(* PLC project Untitled1, Beckhoff Automation GmbH TwinCAT PLC Control 3.5.13.21 *)
(* stored: creationDateTime 2024-03-06T00:00:47.2111878, modificationDateTime 2024-03-06T00:00:47.2111878 *)

PROGRAM main_1
VAR
//Problem1: Start from input1, go clockwise(out1) reset from input 3. To have sufficient time to stop, the Reset button will remain 
//active for 3s from Tof_0. The condition to reset out1 is that out1 has to be active, and out2 has to deactivate. 
//The condition to active out1 is out2 has to deactivate, reset for out1 and out2 has to deactive. The same thing for out2 go for counterclockwise


//Problem2 :Start from input1, it will active Tof_2 for 5 seconds -> run out1 from RS_0 for 5 seconds. And out1 connect to ToN_0, so it 
//will hold ton_0 for 5s at the same time. After hold ton_0 for 5s, it will active tof_3 (hold 3s to active ton_1 -> active tof_4 to run 
//out2 for 4s) )and tof_7 (reset rs_0-> turn off out1) at the same time. So tof3 and ton1 is use for stop out1 for 3s.
//After out2 run FOR 4S, it will active ton2 ->reset  out2 AND tof5 active AND hold 3S TO active ton3 (3S stop FOR out2). After ton3 
//active it will start the loop again because it connects TO set OF rs0.
//Condition to start out1 is non of them(out1,out2) is reseting(cooldown), input3 is not press
//Condition to reset out1 is out1 is running and out 2 is not running, input3 is pressed.
//Same condition to reset out2


//Problem3: Input1 start sr7 TO run out1. Sensor1 active will stop out1 AND active tof6 FOR 3S AND hold ton4 FOR 3S 
//(3s break after change direction) -> out2 run. Sensor 2 active will reset out1 and do the same thing as sensor 1 to run out1
//Condition TO run out1, out2 BY sensor is only 1 sensor is active AT the same TIME. Sr6 AND sr4 are use TO make sure out1, 
//out1 are only active by sensor after we start out1 with input1. 
//Condition under input1 is to make sure input1 cannot affect tonthe process when changing direction by sensors.
//Condition to reset is same as problem 1.


	//IMPORTANCE: ADD NEGATION TO ALL INPUT 3 BEFORE RUN IN REAL PLC. Deactive other problems when run one.
	input1 AT %I* : BOOL; //sj1
	out1 AT %Q* : BOOL; // clockwise
	
	input2 AT %I* : BOOL; //sj2
	out2 AT %Q* : BOOL; // counterclockwise
	
	input3 AT %I* : BOOL; //sj3
	sensor1 AT %I* : BOOL; //sensor1
	sensor2 AT %I* : BOOL; //sensor2
	
	SR_0: sr;
	start: BOOL;
	stop: BOOL;
	SR_1: sr;
	stop1: BOOL;
	timer1: TON;
	out3: BOOL;
	TimV: TIME;
	tim1out: BOOL;
	timer2: TON;
	SR_2: sr;
	tim2out: BOOL;
	timer3: TON;
	timer4: TON;
	TOF_0: TOF;
	TOF_1: TOF;
	TOF_2: TOF;
	TOF_3: TOF;
	TON_0: TON;
	TON_1: TON;
	TOF_4: TOF;
	SR_3: sr;
	TON_2: TON;
	TOF_5: TOF;
	TON_3: TON;
	SR_4: sr;
	TON_4: TON;
	TOF_6: TOF;
	SR_5: SR;
	SR_6: SR;
	TOF_7: TOF;
	TON_5: TON;
	SR_7: SR;
	TOF_8: TOF;
	TOF_9: TOF;
	TOF_10: TOF;
	RS_0: RS;
	RS_1: RS;
	test: BOOL;
	TON_6: ton;
	SR_8: sr;
END_VAR

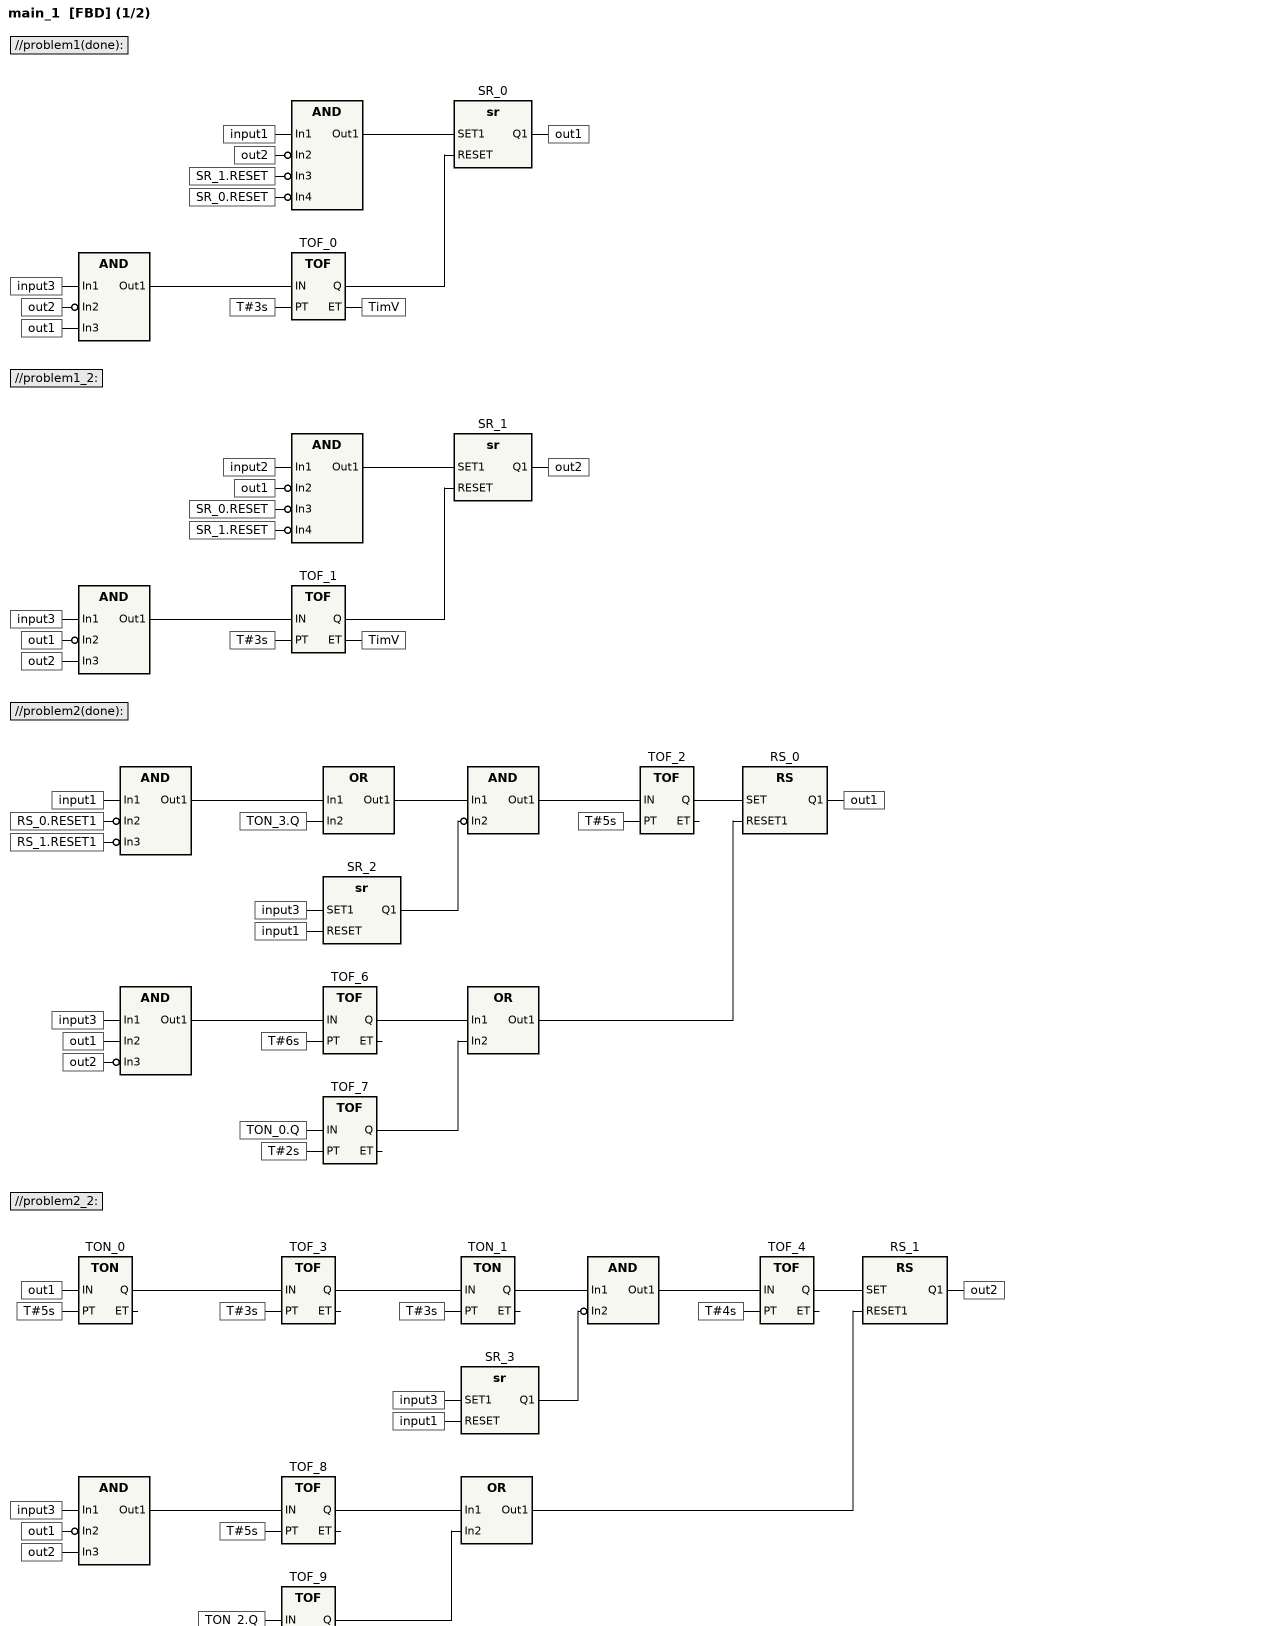
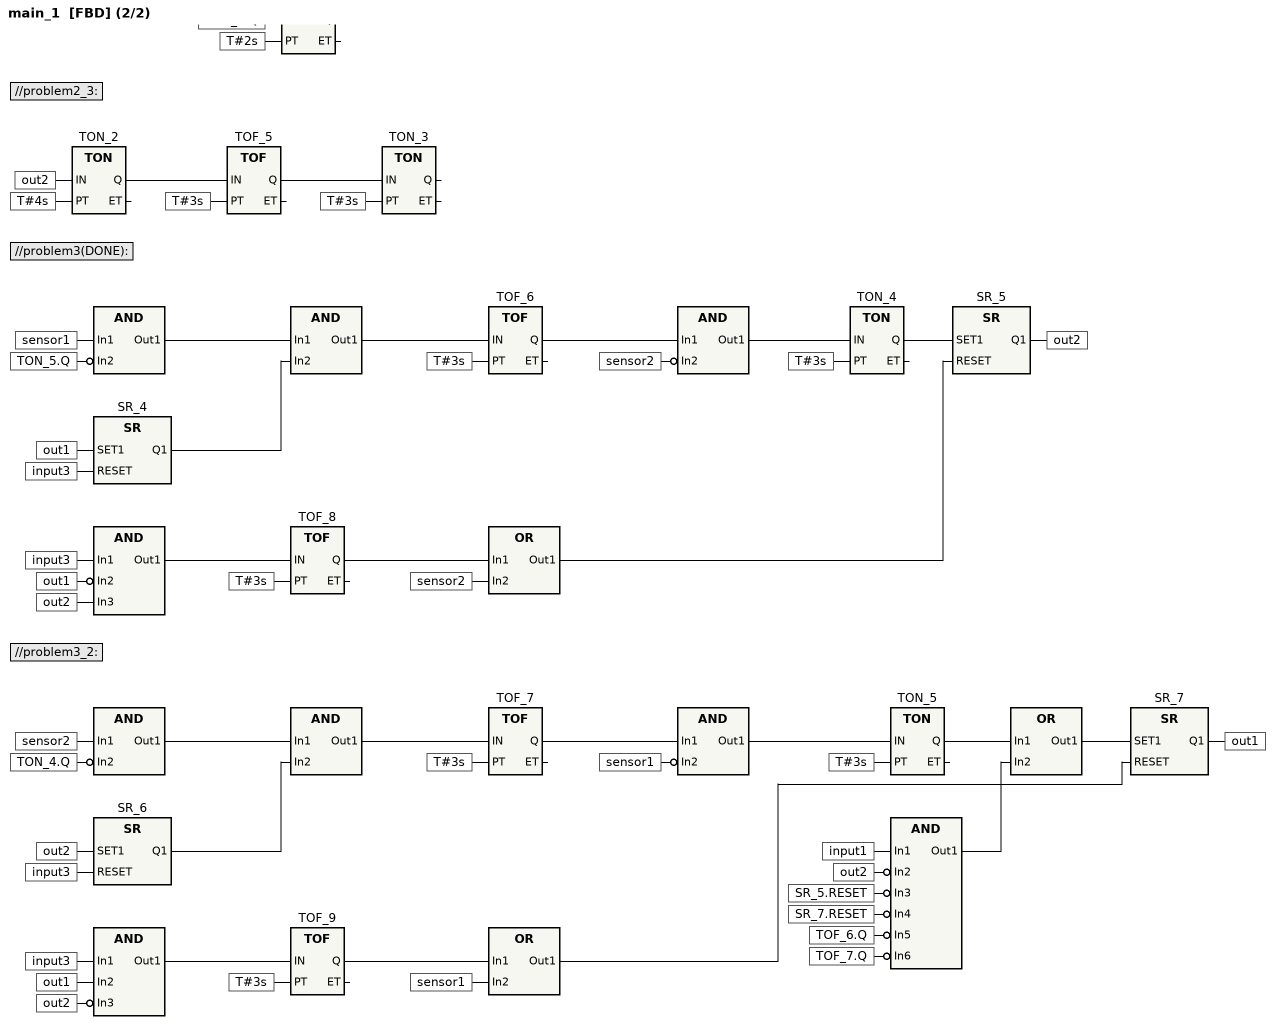
(* FBD diagram, written out as Structured Text *)
//problem1(done):
TOF_0(IN := input3 AND NOT out2 AND out1, PT := T#3s, ET => TimV);
SR_0(SET1 := input1 AND NOT out2 AND NOT SR_1.RESET AND NOT SR_0.RESET, RESET := TOF_0.Q);
out1 := SR_0.Q1;
//problem1_2:
TOF_1(IN := input3 AND NOT out1 AND out2, PT := T#3s, ET => TimV);
SR_1(SET1 := input2 AND NOT out1 AND NOT SR_0.RESET AND NOT SR_1.RESET, RESET := TOF_1.Q);
out2 := SR_1.Q1;
//problem2(done):
SR_2(SET1 := input3, RESET := input1);
TOF_2(IN := (input1 AND NOT RS_0.RESET1 AND NOT RS_1.RESET1 OR TON_3.Q) AND NOT SR_2.Q1, PT := T#5s);
TOF_6(IN := input3 AND out1 AND NOT out2, PT := T#6s);
TOF_7(IN := TON_0.Q, PT := T#2s);
RS_0(SET := TOF_2.Q, RESET1 := TOF_6.Q OR TOF_7.Q);
out1 := RS_0.Q1;
//problem2_2:
TON_0(IN := out1, PT := T#5s);
TOF_3(IN := TON_0.Q, PT := T#3s);
TON_1(IN := TOF_3.Q, PT := T#3s);
SR_3(SET1 := input3, RESET := input1);
TOF_4(IN := TON_1.Q AND NOT SR_3.Q1, PT := T#4s);
TOF_8(IN := input3 AND NOT out1 AND out2, PT := T#5s);
TOF_9(IN := TON_2.Q, PT := T#2s);
RS_1(SET := TOF_4.Q, RESET1 := TOF_8.Q OR TOF_9.Q);
out2 := RS_1.Q1;
//problem2_3:
TON_2(IN := out2, PT := T#4s);
TOF_5(IN := TON_2.Q, PT := T#3s);
TON_3(IN := TOF_5.Q, PT := T#3s);
//problem3(DONE):
SR_4(SET1 := out1, RESET := input3);
TOF_6(IN := sensor1 AND NOT TON_5.Q AND SR_4.Q1, PT := T#3s);
TON_4(IN := TOF_6.Q AND NOT sensor2, PT := T#3s);
TOF_8(IN := input3 AND NOT out1 AND out2, PT := T#3s);
SR_5(SET1 := TON_4.Q, RESET := TOF_8.Q OR sensor2);
out2 := SR_5.Q1;
//problem3_2:
SR_6(SET1 := out2, RESET := input3);
TOF_7(IN := sensor2 AND NOT TON_4.Q AND SR_6.Q1, PT := T#3s);
TON_5(IN := TOF_7.Q AND NOT sensor1, PT := T#3s);
TOF_9(IN := input3 AND out1 AND NOT out2, PT := T#3s);
SR_7(SET1 := TON_5.Q OR input1 AND NOT out2 AND NOT SR_5.RESET AND NOT SR_7.RESET AND NOT TOF_6.Q AND NOT TOF_7.Q, RESET := TOF_9.Q OR sensor1);
out1 := SR_7.Q1;
END_PROGRAM
